# B&R Automation Studio project X20CP1586AS4SHA256
Automation Studio 4.12.5.95 SP

## Configuration Config1

CPU X20CP1586, AutomationRuntime B4.93, Build 4.1.2, Vc V4.72.6

### Task classes (Cpu.sw)
```
Cyclic#1 (cycle 1000000 us, tolerance 0 us):
  CycleTime <- CycleTime.prg
  SHA256 <- SHA256.prg
  Program <- (binary)
Binaries: udbdef, FWRules, TCData, iomap, ashwac, Role, sysconf, arconfig, asfw, User, ashwd
Libraries: runtime, astime, asieccon
```

### Hardware
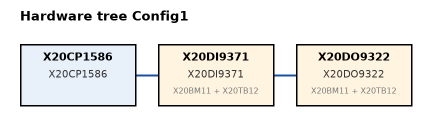
```
X20BM11 : X20BM11 v1.1.0.0  [X2X1 -> X20CP1586.IF6]
X20BM11a : X20BM11 v1.1.0.0  [X2X1 -> X20BM11.X2X2]
X20CP1586 : X20CP1586 v1.10.0.0
  Connector IF2:
    ActivateDevice = 1
  ConfigurationID = X20CP1586AS4_Config1
  SystemTick = 100
  TaskClassIdleTime = 400
  CyclicTaskClassCount = 2
  Cyclic1Duration = 1000000
  Cyclic1Tolerance = 0
  Cyclic2Duration = 1000
  Cyclic2Tolerance = 0
  Cyclic3Duration = 1000
  Cyclic3Tolerance = 1000
  Cyclic4Duration = 100
  Cyclic4Tolerance = 100
  FileDevice1
  FileDeviceName1 = USER
  FileDevicePath1 = USER_PATH
  ActivateSntp = 1
  SntpcServAddr1 = time.google.com
  SntpcServAddr2 = time.aws.com
  SntpcServAddr3 = time.cloudflare.com
  SntpcServAddr4 = time.windows.com
  ActivateOpcUa = 1
  OpcUa_AuthenticationSecurityPolicy_EnableNone = 1
  OpcUa_AuthenticationSecurityPolicy_EnableBasic128Rsa15 = 1
  OpcUaInformationModels_PV_Version = 1
X20DI9371 : X20DI9371 v1.4.0.0  [SS1 -> X20TB12.SS; SL -> X20BM11.SL1]
X20DO9322 : X20DO9322 v1.5.0.0  [SS1 -> X20TB12a.SS; SL -> X20BM11a.SL1]
X20TB12 : X20TB12 v1.0.0.0
X20TB12a : X20TB12 v1.0.0.0
```

### IoMap.iom - X20CP1586/IoMap.iom
```iecst
VAR_CONFIG
	::LED12 AT %QX."X20DO9322".DigitalOutput12;
	::LED11 AT %QX."X20DO9322".DigitalOutput11;
END_VAR
```

## Logical view

### Global.var - Global variables
```iecst
VAR
	LED11 : {REDUND_UNREPLICABLE} BOOL;
	LED12 : {REDUND_UNREPLICABLE} BOOL := TRUE;
END_VAR
```

### Program Logical/BlinkerL (IEC)

#### Cyclic.ld
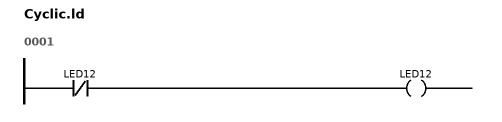
Ladder, written as Structured Text:
```iecst
PROGRAM _CYCLIC
(* Network 1 *)
LED12 := NOT LED12;
END_PROGRAM
```

### Program Logical/SHA256 (ANSIC)

#### Main.c - Init, cyclic, exit code
```c
#include <bur/plctypes.h>
#include <inttypes.h>

#ifdef _DEFAULT_INCLUDES
#include <AsDefault.h>
#endif

#include "sha256.h"

uint64_t rdtsc() {
	uint32_t low, high;
	__asm__ __volatile__(
	"rdtsc"
	: "=a" (low),
	"=d" (high)
	);
		return ((uint64_t)high << 32) | low;
}

static long long begin, begin_saved, end;

void _INIT ProgramInit(void)
{
	int i; //C99
	for(i = 0; i< sizeof(buffer); i++) buffer[i] = 'a';
}

void _CYCLIC ProgramCyclic(void)
{
	SHA256_CTX ctx;

	begin = rdtsc();
	cycle_time = (LREAL)(begin - begin_saved);
	begin_saved = begin;

	sha256_init(&ctx);
	sha256_update(&ctx, buffer, sizeof(buffer));
	sha256_final(&ctx, digest);

	end = rdtsc();
	cpu_time_used = ((LREAL)(end - begin));

	MBperSec = cycle_time / cpu_time_used;
}

void _EXIT ProgramExit(void) {}
```

#### sha256.c
```c
/******************************************************************************
* Filename:   sha256.c
* Author:     Brad Conte (brad AT bradconte.com)
* Copyright:
* Disclaimer: This code is presented "as is" without any guarantees.
* Details:    Implementation of the SHA-256 hashing algorithm.
              SHA-256 is one of the three algorithms in the SHA2
              specification. The others, SHA-384 and SHA-512, are not
              offered in this implementation.
Algorithm specification can be found here:
http://csrc.nist.gov/publications/fips/fips180-2/fips180-2withchangenotice.pdf
              This implementation uses little endian byte order.
******************************************************************************/

/*************************** HEADER FILES ***************************/
//#include <ansi_c.h>
#include <stdlib.h>
//#include <memory.h>
#include "sha256.h"

/****************************** MACROS ******************************/
#define ROTLEFT(a,b) (((a) << (b)) | ((a) >> (32-(b))))
#define ROTRIGHT(a,b) (((a) >> (b)) | ((a) << (32-(b))))

#define CH(x,y,z) (((x) & (y)) ^ (~(x) & (z)))
#define MAJ(x,y,z) (((x) & (y)) ^ ((x) & (z)) ^ ((y) & (z)))
#define EP0(x) (ROTRIGHT(x,2) ^ ROTRIGHT(x,13) ^ ROTRIGHT(x,22))
#define EP1(x) (ROTRIGHT(x,6) ^ ROTRIGHT(x,11) ^ ROTRIGHT(x,25))
#define SIG0(x) (ROTRIGHT(x,7) ^ ROTRIGHT(x,18) ^ ((x) >> 3))
#define SIG1(x) (ROTRIGHT(x,17) ^ ROTRIGHT(x,19) ^ ((x) >> 10))

/**************************** VARIABLES *****************************/
static const unsigned int k[64] = {
	0x428a2f98,0x71374491,0xb5c0fbcf,0xe9b5dba5,0x3956c25b,0x59f111f1,0x923f82a4,0xab1c5ed5,
	0xd807aa98,0x12835b01,0x243185be,0x550c7dc3,0x72be5d74,0x80deb1fe,0x9bdc06a7,0xc19bf174,
	0xe49b69c1,0xefbe4786,0x0fc19dc6,0x240ca1cc,0x2de92c6f,0x4a7484aa,0x5cb0a9dc,0x76f988da,
	0x983e5152,0xa831c66d,0xb00327c8,0xbf597fc7,0xc6e00bf3,0xd5a79147,0x06ca6351,0x14292967,
	0x27b70a85,0x2e1b2138,0x4d2c6dfc,0x53380d13,0x650a7354,0x766a0abb,0x81c2c92e,0x92722c85,
	0xa2bfe8a1,0xa81a664b,0xc24b8b70,0xc76c51a3,0xd192e819,0xd6990624,0xf40e3585,0x106aa070,
	0x19a4c116,0x1e376c08,0x2748774c,0x34b0bcb5,0x391c0cb3,0x4ed8aa4a,0x5b9cca4f,0x682e6ff3,
	0x748f82ee,0x78a5636f,0x84c87814,0x8cc70208,0x90befffa,0xa4506ceb,0xbef9a3f7,0xc67178f2
};

/*********************** FUNCTION DEFINITIONS ***********************/
void sha256_transform(SHA256_CTX *ctx, const USINT data[])
{
	unsigned int a, b, c, d, e, f, g, h, i, j, t1, t2, m[64] = {0};

	for (i = 0, j = 0; i < 16; ++i, j += 4)
		m[i] = (data[j] << 24) | (data[j + 1] << 16) | (data[j + 2] << 8) | (data[j + 3]);
	for ( ; i < 64; ++i)
		m[i] = SIG1(m[i - 2]) + m[i - 7] + SIG0(m[i - 15]) + m[i - 16];

	a = ctx->state[0];
	b = ctx->state[1];
	c = ctx->state[2];
	d = ctx->state[3];
	e = ctx->state[4];
	f = ctx->state[5];
	g = ctx->state[6];
	h = ctx->state[7];

	for (i = 0; i < 64; ++i) {
		t1 = h + EP1(e) + CH(e,f,g) + k[i] + m[i];
		t2 = EP0(a) + MAJ(a,b,c);
		h = g;
		g = f;
		f = e;
		e = d + t1;
		d = c;
		c = b;
		b = a;
		a = t1 + t2;
	}

	ctx->state[0] += a;
	ctx->state[1] += b;
	ctx->state[2] += c;
	ctx->state[3] += d;
	ctx->state[4] += e;
	ctx->state[5] += f;
	ctx->state[6] += g;
	ctx->state[7] += h;
}

void sha256_init(SHA256_CTX *ctx)
{
	ctx->datalen = 0;
	ctx->bitlen = 0;
	ctx->state[0] = 0x6a09e667;
	ctx->state[1] = 0xbb67ae85;
	ctx->state[2] = 0x3c6ef372;
	ctx->state[3] = 0xa54ff53a;
	ctx->state[4] = 0x510e527f;
	ctx->state[5] = 0x9b05688c;
	ctx->state[6] = 0x1f83d9ab;
	ctx->state[7] = 0x5be0cd19;
}

void sha256_update(SHA256_CTX *ctx, const USINT data[], size_t len)
{
	unsigned int i;

	for (i = 0; i < len; ++i) {
		ctx->data[ctx->datalen] = data[i];
		ctx->datalen++;
		if (ctx->datalen == 64) {
			sha256_transform(ctx, ctx->data);
			ctx->bitlen += 512;
			ctx->datalen = 0;
		}
	}
}

void sha256_final(SHA256_CTX *ctx, USINT hash[])
{
	unsigned int i, j;

	i = ctx->datalen;

	// Pad whatever data is left in the buffer.
	if (ctx->datalen < 56) {
		ctx->data[i++] = 0x80;
		while (i < 56)
			ctx->data[i++] = 0x00;
	}
	else {
		ctx->data[i++] = 0x80;
		while (i < 64)
			ctx->data[i++] = 0x00;
		sha256_transform(ctx, ctx->data);
		for (j = 0; j < 56; j++) ctx->data[j] = 0;
		//memset(ctx->data, 0, 56);
	}

	// Append to the padding the total message's length in bits and transform.
	ctx->bitlen += ctx->datalen * 8;
	ctx->data[63] = (USINT)(ctx->bitlen);
	ctx->data[62] = (USINT)(ctx->bitlen >> 8);
	ctx->data[61] = (USINT)(ctx->bitlen >> 16);
	ctx->data[60] = (USINT)(ctx->bitlen >> 24);
	ctx->data[59] = (USINT)(ctx->bitlen >> 32);
	ctx->data[58] = (USINT)(ctx->bitlen >> 40);
	ctx->data[57] = (USINT)(ctx->bitlen >> 48);
	ctx->data[56] = (USINT)(ctx->bitlen >> 56);
	sha256_transform(ctx, ctx->data);

	// Since this implementation uses little endian byte ordering and SHA uses big endian,
	// reverse all the bytes when copying the final state to the output hash.
	for (i = 0; i < 4; ++i) {
		hash[i]      = (ctx->state[0] >> (24 - i * 8)) & 0x000000ff;
		hash[i + 4]  = (ctx->state[1] >> (24 - i * 8)) & 0x000000ff;
		hash[i + 8]  = (ctx->state[2] >> (24 - i * 8)) & 0x000000ff;
		hash[i + 12] = (ctx->state[3] >> (24 - i * 8)) & 0x000000ff;
		hash[i + 16] = (ctx->state[4] >> (24 - i * 8)) & 0x000000ff;
		hash[i + 20] = (ctx->state[5] >> (24 - i * 8)) & 0x000000ff;
		hash[i + 24] = (ctx->state[6] >> (24 - i * 8)) & 0x000000ff;
		hash[i + 28] = (ctx->state[7] >> (24 - i * 8)) & 0x000000ff;
	}
}
```

#### sha256.h
```c
/*********************************************************************
* Filename:   sha256.h
* Author:     Brad Conte (brad AT bradconte.com)
* Copyright:
* Disclaimer: This code is presented "as is" without any guarantees.
* Details:    Defines the API for the corresponding SHA1 implementation.
*********************************************************************/

#ifndef SHA256_H
#define SHA256_H

/*************************** HEADER FILES ***************************/
#include <stddef.h>
#include <bur/plctypes.h>

/****************************** MACROS ******************************/
#define SHA256_BLOCK_SIZE 32            // SHA256 outputs a 32 byte digest

/**************************** DATA TYPES ****************************/
// typedef unsigned char BYTE;             // 8-bit byte
// typedef unsigned int  WORD;             // 32-bit word, change to "long" for 16-bit machines

typedef struct {
	USINT data[64];
	unsigned int datalen;
	unsigned long long bitlen;
	unsigned int state[8];
} SHA256_CTX;

/*********************** FUNCTION DECLARATIONS **********************/
void sha256_init(SHA256_CTX *ctx);
void sha256_update(SHA256_CTX *ctx, const USINT data[], size_t len);
void sha256_final(SHA256_CTX *ctx, USINT hash[]);

#endif   // SHA256_H
```

#### Variables.var - Local variables
```iecst
VAR
	digest : ARRAY[0..31] OF USINT;
	buffer : ARRAY[0..1048575] OF USINT;
	cpu_time_used : LREAL;
	cycle_time : LREAL;
	cycles_counter : UDINT;
	MBperSec : LREAL;
END_VAR
```

### Program Logical/BlinkerC (ANSIC)

#### Main.c
```c
#include <bur/plctypes.h>

#ifdef _DEFAULT_INCLUDES
	#include <AsDefault.h>
#endif

void _INIT ProgramInit(void)
{

}

void _CYCLIC ProgramCyclic(void)
{
	LED11 =  !LED11;
}

void _EXIT ProgramExit(void)
{

}
```

### Program Logical/CycleTime (ANSIC)

#### Variables.var
```iecst
VAR
	CycleTimeTicks : UDINT;
END_VAR
```

#### Main.c
```c
#include <bur/plctypes.h>
#include <inttypes.h>

#ifdef _DEFAULT_INCLUDES
	#include <AsDefault.h>
#endif

static uint64_t cycles, cycles_saved;

uint64_t rdtsc() {
	uint32_t low, high;
	__asm__ __volatile__(
		"rdtsc"
		: "=a" (low),
		"=d" (high)
	);
	return ((uint64_t)high << 32) | low;
}

void _INIT ProgramInit(void)
{
	cycles_saved = rdtsc();

}

void _CYCLIC ProgramCyclic(void)
{
	cycles = rdtsc();
	CycleTimeTicks = (UDINT)(cycles - cycles_saved);
	cycles_saved = cycles;
}

void _EXIT ProgramExit(void) { }
```

Listed in the project but not available here: Logical/Global.typ, Logical/Libraries, Logical/SHA256/Types.typ
